TYPE UValues :
UNION
	Binary: BOOL;
	Numeric: LREAL;
	String_t: STRING;
END_UNION
END_TYPE

(* stored: Version 1.1.0.1, ProductVersion 3.1.4024.9
   DUT UValues: Id {eab437b1-daf4-43d1-8d5d-d652d94538e5} *)
